FUNCTION_BLOCK Tank_SystemOff EXTENDS _Tank_State IMPLEMENTS I_Execute
VAR
	_exe			: Execute(THIS^);
END_VAR

METHOD Execute
IF _ctx.priv.iIsSystemOn.IsLowered() THEN
	IF _ctx.priv.smgr.Current <> _ctx.state.iSystemOff THEN
		_ctx.priv.smgr.Request(_ctx.state.iSystemOff);
	END_IF
END_IF
END_METHOD

METHOD OnExecute
IF _ctx.priv.iIsSystemOn.IsRised() THEN
	IF _ctx.priv.smgr.Current = _ctx.state.iSystemOff THEN
		_ctx.priv.smgr.Request(_ctx.state.iDisabled);
	END_IF
END_IF
END_METHOD

METHOD OnInit
_ctx.io.out.bInletValveOpen := FALSE;
_ctx.hmi.bResetButtonVis := FALSE;
_ctx.priv.IsFillable.Rise();
END_METHOD

END_FUNCTION_BLOCK

(* stored: Version 1.1.0.1
   POU Tank_SystemOff: Id {2f202dd8-f0b6-4b76-ae64-f34cbab5f204}, SpecialFunc None
   Method Execute: Id {321e3024-2b6e-4235-8d48-c94d4f0858d3}
   Method OnExecute: Id {10ccc01f-0593-48d1-ad6e-86730bf47ac1}
   Method OnInit: Id {56d030fd-7ae1-4166-b892-6183b53d27ee} *)
